(* CoDeSys 2.3 export: MNG_SIMULATION.EXP *)

(* POU MNG_Simulation, ST *)
FUNCTION_BLOCK MNG_Simulation
VAR_INPUT
    bEnable    : BOOL                          := FALSE;
    outputs    : MNG_Application_Outputs_32Bit         ;
END_VAR
VAR_OUTPUT
    inputs     : MNG_Application_Inputs_32Bit          ;
END_VAR
VAR
    ioUpdater  : MNG_UpdateIOs                 := (sRemoteHost := '127.0.0.1', nRemotePort := 6001);
    fbCloseAll : FB_SocketCloseAll;
    bCloseAll  : BOOL := TRUE;
END_VAR
IF bCloseAll THEN (*On PLC reset or program download close all old (opened) connections *)
    bCloseAll := FALSE;
    fbCloseAll( bExecute:= TRUE );
ELSE
    fbCloseAll( bExecute:= FALSE );
END_IF

IF NOT fbCloseAll.bBusy THEN

    (* ------------------------------------- trigger data exchange ----------------------------------------------------------------------------*)
    ioUpdater(Outputs := outputs, Inputs => inputs, bEnable := bEnable);

END_IF

END_FUNCTION_
END_FUNCTION_BLOCK
